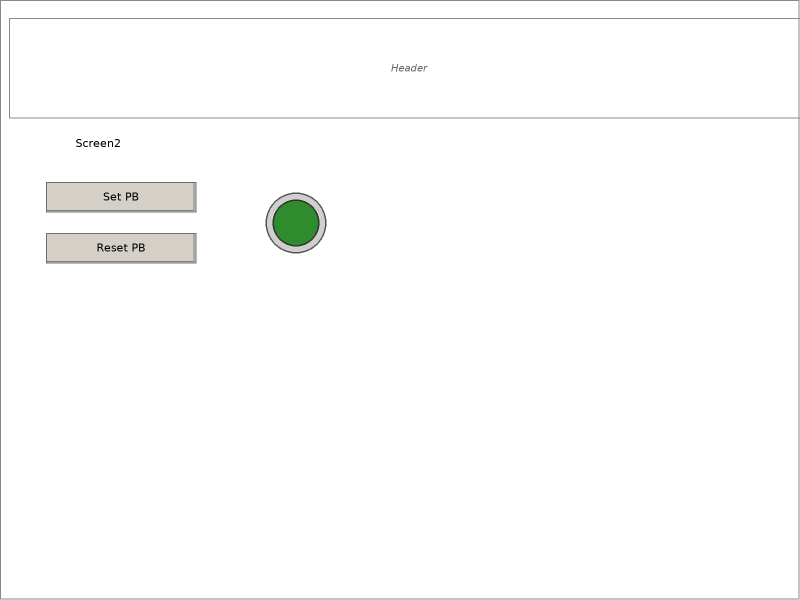
VISUALIZATION Screen2  // 800x600
    Label (46,110 105x67), "Screen2"
    Button (46,182 150x30), "Set PB", colour toggle: GVL.Bool1
        tap GVL.Bool1
    Lamp1 (261,188 70x70), variable: GVL.Bool3, style: Lamp-Lamp1-Green
    Button (46,233 150x30), "Reset PB", colour toggle: GVL.Bool2
        tap GVL.Bool2
    Frame (9,18 800x100)
        shows Header()
END_VISUALIZATION

(* stored: Version 1.1.0.1, ProductVersion 3.1.4024.12
   Visu Screen2: Id {2d751ee3-0b7d-4357-8e6a-921625746514} *)
